INTERFACE ITF_LimitSwitch

PROPERTY Active : BOOL
GET
END_GET
SET
END_SET
END_PROPERTY

METHOD Update : BOOL
VAR_INPUT
	iActive : BOOL;   // TRUE = eindschakelaar aangetikt
END_VAR
END_METHOD

END_INTERFACE

(* stored: Version 1.1.0.1
   Itf ITF_LimitSwitch: Id {ed133e1e-cddc-499f-baad-80792598d895}
   Property Active: Id {5718ee03-d12b-4cde-abf0-f778167646b3}
   Get Get: Id {28578ffb-04d7-44c6-adbd-5939e1986407}
   Set Set: Id {817f20ea-ac9e-4c0a-bef0-3d2245750fe5}
   Method Update: Id {86c43624-59b7-4b74-909a-435d308aef2e} *)
